// Valid on Done (S3.10).
TYPE ST_StaubliConnOutCmd :
STRUCT
    Reconnected    : BOOL;
    ControllerCode : STRING(64);   // the robot's own last error code, if any
END_STRUCT
END_TYPE

(* stored: Version 1.1.0.1, ProductVersion 3.1.4024.12
   DUT ST_StaubliConnOutCmd: Id {eb90a33a-1f28-4ce4-a590-a2cc71a8a5f3} *)
